// TIA Portal V20 export
TYPE "typeDataFromSafety"
// stored: Access Published, IsFailsafeCompliant true, Namespace Safety
   STRUCT
      devicesSummary { ExternalWritable := 'False'} : "Safety.typeDevicesStatusSummary";   // General safety status of devices
      mainOp { ExternalWritable := 'False'} : "Safety.typeMainOpMode";   // Main Op State
      pHmi { ExternalWritable := 'False'} : "Safety.typePhmi";   // Phmi State
      scsMode { ExternalWritable := 'False'} : "Safety.typeScsMode";   // SCS Mode
      rcMode1 { ExternalWritable := 'False'} : "Safety.typeRollChangeMode";   // LH Roll Change State
      rcMode2 { ExternalWritable := 'False'} : "Safety.typeRollChangeMode";   // RH Roll Change State
      scrapBox1 { ExternalWritable := 'False'} : "Safety.typeScrapBoxCommands";   // Scrap Box Command
      eStopStatus { ExternalWritable := 'False'} : "Safety.typeEstopStatus";   // E Stop Pressed
      fDoorSwitchStatus { ExternalWritable := 'False'} : "Safety.typeFDoorSwitchStatus";   // F Door Open Status
      fDoorCoilStatus { ExternalWritable := 'False'} : "Safety.typeFDoorUnlockOutput";   // F Door Unlock Cmd Status
      Zone1SafetyOpEnable { ExternalWritable := 'False'} : "Safety.typeSafetyOperationEnable";   // Zone1 Operation Enable
      Zone2SafetyOpEnable { ExternalWritable := 'False'} : "Safety.typeSafetyOperationEnable";   // Zone2 Operation Enable
      Zone3SafetyOpEnable { ExternalWritable := 'False'} : "Safety.typeSafetyOperationEnable";   // Zone3 Operation Enable
      eStopZone1 { ExternalWritable := 'False'} : "Safety.typeEstopFunction";   // Safety status of estop button in Zone.1
      eStopZone2 { ExternalWritable := 'False'} : "Safety.typeEstopFunction";   // Safety status of estop button in Zone.2
      eStopZone3 { ExternalWritable := 'False'} : "Safety.typeEstopFunction";   // Safety status of estop button in Zone.3
      statusZone1 { ExternalWritable := 'False'} : "Safety.typeSafetyZoneStatus";   // Status of safety zone
      statusZone2 { ExternalWritable := 'False'} : "Safety.typeSafetyZoneStatus";   // Status of safety zone
      statusZone3 { ExternalWritable := 'False'} : "Safety.typeSafetyZoneStatus";   // Status of safety zone
      fDoorDrive { ExternalWritable := 'False'} : "Safety.typeFDoorFunction";
      driveStatus { ExternalWritable := 'False'} : "Safety.typeSafetyDriveStatus";
      safetySensor { ExternalWritable := 'False'} : "Safety.typeSafetySensor";
      feedbackFault { ExternalWritable := 'False'} : "Safety.typeFeedbackFault";
      radiusStatus { ExternalWritable := 'False'} : "Safety.typeRadiusStatusSummary";
      cvCoverStatus { ExternalWritable := 'False'} : "Safety.typeCvCoverStatus";
      EnableACK { ExternalWritable := 'False'} : Bool;
      SS1Extention { ExternalWritable := 'False'} : Bool;
      LHSS1Extenstion { ExternalWritable := 'False'} : Bool;
      RHSS1Extenstion { ExternalWritable := 'False'} : Bool;
      AllEstopsOK { ExternalWritable := 'False'} : Bool;   // E Stop On Station All Ok
      Z_Fold_AllEstopsOK { ExternalWritable := 'False'} : Bool;   // Z-FOLD System All EMO OK
      AllFdoorClose { ExternalWritable := 'False'} : Bool;   // F Door All Closed
      AllSFDoorOpen { ExternalWritable := 'False'} : Bool;   // F Door Single Open
      AnyNoMFDoorOpen { ExternalWritable := 'False'} : Bool;   // F Door No Multi Open
      safetyReleasedAllSafetyZones { ExternalWritable := 'False'} : Bool := false;   // All safety zones are released
      ackRequiredAnySafetyZone { ExternalWritable := 'False'} : Bool := false;   // At least one safety zone requires an acknowledge
      ackOP_changeRequired { ExternalWritable := 'False'} : Bool := false;   // ACK_OP is waiting for value change
      ackOperatorControlCondition { ExternalWritable := 'False'} : Bool;   // Ack Hmi Oprating Possible
      doorBoxAllReset { ExternalWritable := 'False'} : Bool;   // Combine All Door Box Reset Button
      totalSafetyReset { ExternalWritable := 'False'} : Bool;   // Combine All Reset Trigger
      zone1DoorOpenRequest { ExternalWritable := 'False'} : Bool;   // Zone 1 Door Open Request
      zone2DoorOpenRequest { ExternalWritable := 'False'} : Bool;   // Zone 2 Door Open Request
      zone3DoorOpenRequest { ExternalWritable := 'False'} : Bool;   // Zone 3 Door Open Request
      zone1DriveAckReq { ExternalWritable := 'False'} : Bool;   // Zone 1 Safety Fault Ack Request
      zone2DriveAckReq { ExternalWritable := 'False'} : Bool;   // Zone 2 Safety Fault Ack Request
      zone3DriveAckReq { ExternalWritable := 'False'} : Bool;   // Zone 3 Safety Fault Ack Request
      noSafetyFault { ExternalWritable := 'False'} : Bool;   // All Zone No Safety Fault
      connectionBoxID { ExternalWritable := 'False'} : Int;   // PHmi Connection Box ID
      no_Corver_RC { ExternalWritable := 'False'} : Bool;   // Not detected Frame Corver In Roll Change
      LH_RollChangeActive { ExternalWritable := 'False'} : Bool;
      RH_RollChangeActive { ExternalWritable := 'False'} : Bool;
      FrameCoverNG { ExternalWritable := 'False'} : Bool;   // FrameCover Not Detect
      BA30CathodeCoverClose { ExternalAccessible := 'False'; ExternalVisible := 'False'; ExternalWritable := 'False'} : Bool;
      BA30AnodeCoverClose { ExternalAccessible := 'False'; ExternalVisible := 'False'; ExternalWritable := 'False'} : Bool;
      BA40CathodeCoverClose { ExternalAccessible := 'False'; ExternalVisible := 'False'; ExternalWritable := 'False'} : Bool;
      BA40AnodeCoverClose { ExternalAccessible := 'False'; ExternalVisible := 'False'; ExternalWritable := 'False'} : Bool;
      BA60ExternalDoorOpen { ExternalAccessible := 'False'; ExternalVisible := 'False'; ExternalWritable := 'False'} : Bool;
      BA60jrPPLeftDoorForcedOpen { ExternalAccessible := 'False'; ExternalVisible := 'False'; ExternalWritable := 'False'} : Bool;
      BA60jrPPLeftDoorNormalOpen { ExternalAccessible := 'False'; ExternalVisible := 'False'; ExternalWritable := 'False'} : Bool;
      BA60Stacker1LightCurtainDetect : Bool;
      BA60Stacker2LightCurtainDetect { ExternalAccessible := 'False'; ExternalVisible := 'False'; ExternalWritable := 'False'} : Bool;
      BA60Stacker2MaintanceDoorNormalOpen { ExternalAccessible := 'False'; ExternalVisible := 'False'; ExternalWritable := 'False'} : Bool;
      BA60Stacker2MaintanceDoorForcedOpen { ExternalAccessible := 'False'; ExternalVisible := 'False'; ExternalWritable := 'False'} : Bool;
      FdoorLamp : "Safety.fDoorLamp";
      DoorBoxUnlockSW : "Safety.typeDoorUnlockSW";
      BA015 { ExternalWritable := 'False'} : "Safety.s_PLC_Interlocks";
      BA030 { ExternalWritable := 'False'} : "Safety.s_PLC_Interlocks";
      BA040 { ExternalWritable := 'False'} : "Safety.s_PLC_Interlocks";
      BA060 { ExternalWritable := 'False'} : "Safety.s_PLC_Interlocks";
   END_STRUCT;
END_TYPE
